(* IEC 61131-3 sources: Automation/pous/functions, 5 files *)

(* ---- Calculate_err.st ---- *)
(* Finds diffrence between desired and actual value *)

FUNCTION Calculate_err : REAL
  VAR_INPUT
    Setpoint : REAL;
    Process_Value : REAL;
  END_VAR

Calculate_err := Setpoint - Process_Value;

END_FUNCTION

(* ---- Engineering_Unit.st ---- *)
(* Applies multiplication factor and offset to a value *)

FUNCTION Engineering_Unit : REAL
  VAR_INPUT
    Value : REAL;
    Unit_Factor : REAL;
    Unit_Offset : REAL;
  END_VAR

Engineering_Unit := (Value * Unit_Factor) + Unit_Offset;

END_FUNCTION

(* ---- Limit_Value.st ---- *)
(* Keeps input vaule from going out of bounds *)

FUNCTION Limit_Value : REAL
  VAR_INPUT
    Value : REAL;
    Min_Value : REAL;
    Max_Value : REAL;
  END_VAR

IF Value < Min_Value THEN
    Limit_Value := Min_Value;
ELSIF Value > Max_Value THEN
    Limit_Value := Max_Value;
ELSE
    Limit_Value := Value;
END_IF;

END_FUNCTION

(* ---- Scale_analog.st ---- *)
(* Takes input in analog and gives mesurement value *)

FUNCTION Scale_analog : REAL
  VAR_INPUT
    Raw_value : REAL;
    Raw_Min : REAL;
    Raw_Max : REAL;
    Eng_Min : REAL;
    Eng_Max : REAL;
  END_VAR

Scale_Analog := (((Raw_Value - Raw_Min) / (Raw_Max - Raw_Min)) * (Eng_Max - Eng_Min)) + Eng_Min;

END_FUNCTION

(* ---- State_Transition.st ---- *)
FUNCTION State_Transition : INT
  VAR_INPUT
    Current_State : INT;
    Required_State : INT;
    Next_State : INT;
  END_VAR

IF Current_State = Required_State THEN
    State_Transition := Next_State;
ELSE
    State_Transition := Current_State;
END_IF;

END_FUNCTION
